TYPE DUT_Sta :
STRUCT
		Staion:ARRAY[1..gc_uiStationNum] OF  DUT_StaHistory;
END_STRUCT
END_TYPE

(* stored: Version 1.1.0.1, ProductVersion 3.1.4024.9
   DUT DUT_Sta: Id {3ca44ae3-fabf-4f15-ab00-7162967f1dd4} *)
